(* PLC project Unnamed, Unknown Unnamed 1 *)
(* stored: creationDateTime 2024-12-23T18:09:04, modificationDateTime 2024-12-23T23:53:12 *)

PROGRAM program0
  VAR
    S1 : BOOL;  (* Push Button *)
    Actual_Input_Signal : BOOL;  (* Actual Input Signal because S1 is non latching *)
    Cylinder_1 : BOOL;  (* If True,cylinder is extended. *)
    Cylinder_2 : BOOL;  (* If True,cylinder is extended. *)
    Cylinder_3 : BOOL;  (* If True,cylinder is extended. *)
    y : BOOL;  (* If True,cylinder-1 is retracted. *)
    B2 : BOOL;  (* If True,cylinder-1 is extended. *)
    B3 : BOOL;  (* If True,cylinder-2 is retracted. *)
    Reset : BOOL;
    B4 : BOOL;  (* If True,cylinder-2 is extended. *)
    B5 : BOOL;  (* If True,cylinder-3 is retracted. *)
    B6 : BOOL;  (* If True,cylinder-3 is extended. *)
    x : BOOL;
    B7 : BOOL;  (* Signals part in magazine *)
    TON0 : TON;
    CTU0 : CTU;
    CTU1 : CTU;
    TOF0 : TOF;
    CTU2 : CTU;
    TON1 : TON;
  END_VAR
  VAR  (* added by the conversion: wires and edge detectors of the diagram *)
    _XOR14_OUT : BOOL;
    R_TRIG1 : R_TRIG;
    R_TRIG2 : R_TRIG;
    _AND32_OUT : BOOL;
    R_TRIG3 : R_TRIG;
  END_VAR

(* FBD diagram, written out as Structured Text *)
Actual_Input_Signal := S1;
Actual_Input_Signal := NOT Reset;
S1 := Actual_Input_Signal;
B7 := Actual_Input_Signal;
y := B7;
Cylinder_1 := NOT y;
TON0(IN := B2, PT := T#4s);
_XOR14_OUT := B2 XOR TON0.Q;
Cylinder_2 := _XOR14_OUT;
Cylinder_3 := NOT _XOR14_OUT AND TON0.Q AND NOT B6;
R_TRIG1(CLK := Cylinder_3);
CTU0(CU := R_TRIG1.Q, R := S1, PV := 10);
R_TRIG2(CLK := NOT Cylinder_3);
CTU1(CU := R_TRIG2.Q, R := S1, PV := 10);
_AND32_OUT := CTU0.CV > 0 AND CTU1.CV > 0 AND CTU0.CV - CTU1.CV = 0;
TOF0(IN := NOT _AND32_OUT, PT := T#2s);
y := _AND32_OUT = TOF0.Q;
R_TRIG3(CLK := y);
CTU2(CU := R_TRIG3.Q, R := S1, PV := 10);
x := CTU2.Q;
TON1(IN := x, PT := T#30s);
Reset := x XOR TON1.Q;
END_PROGRAM

CONFIGURATION Config0
  RESOURCE Res0 ON PLC
    TASK task0(INTERVAL := T#20ms, PRIORITY := 0);
    PROGRAM instance0 WITH task0 : program0;
  END_RESOURCE
END_CONFIGURATION
